// TIA Portal project "trietRot_Nhat" (V16)

(* hardware
DEVICE "S7-1200 station_1"  S7-1200 Station
   slot 0: "Rack_0"  S7-1200 Rack  Rack  V1.0
   slot 1: "PLC_1"  CPU 1214C AC/DC/Rly  6ES7 214-1BG40-0XB0  V4.4
*)

// ===== PLC "PLC_1"  CPU 1214C AC/DC/Rly =====

VAR_GLOBAL   // PLC tag table "Default tag table"
   "START" AT %M6.0 : Bool;
   "AUTO" AT %M6.1 : Bool;
   "TG1" AT %M1.1 : Bool;
   "TG2" AT %M1.2 : Bool;
   "STOP" AT %M6.2 : Bool;
   "Đèn" AT %Q0.0 : Bool;
   "Băng tải 2" AT %Q0.2 : Bool;
   "Tag_1" AT %M2.0 : Bool;
   "CB4" AT %M2.4 : Bool;
   "Băng tải 1" AT %Q0.1 : Bool;
   "CB3" AT %M2.3 : Bool;
   "Tag_2" AT %MD10 : DWord;
   "Tag_3" AT %M3.0 : Bool;
   "Sản phẩm hiện tại" AT %MW10 : Int;
   "Thiết lập số sản phẩm trong thùng" AT %MW20 : Int;
   "CB1" AT %M2.1 : Bool;
   "CB2" AT %M2.2 : Bool;
   "Bơm" AT %Q0.3 : Bool;
   "Van" AT %Q0.4 : Bool;
   "Clock_Byte" AT %MB0 : Byte;
   "Clock_2Hz" AT %M0.3 : Bool;
   "Clock_1.25Hz" AT %M0.4 : Bool;
   "Clock_1Hz" AT %M0.5 : Bool;
   "Clock_0.625Hz" AT %M0.6 : Bool;
   "Clock_0.5Hz" AT %M0.7 : Bool;
   "Tag_5" AT %M10.0 : Bool;
   "Giá trị lượng nước hiện tại" AT %MW40 : Int;
   "Thiết lập lượng nước cần rót" AT %MW30 : Int;
   "Xilanh1" AT %Q0.5 : Bool;
   "Xilanh2" AT %Q0.6 : Bool;
   "Thiết lập số thùng hàng" AT %MW50 : Int;
   "Số thùng hàng hiện tại" AT %MW60 : Int;
   "TG3" AT %M1.3 : Bool;
   "TG4" AT %M1.4 : Bool;
   "Tag_4" AT %M1.5 : Bool;
   "Tag_6" AT %MW100 : Int;
   "Tag_7" AT %M1.6 : Bool;
   "CB5" AT %M2.5 : Bool;
   "Tag_9" AT %M11.0 : Bool;
   "Tag_10" AT %M11.1 : Bool;
   "Tag_11" AT %M12.0 : Bool;
   "Tag_12" AT %M12.1 : Bool;
END_VAR

// folder: System blocks/Program resources

DATA_BLOCK "IEC_Counter_0_DB"   // DB1
{ S7_Optimized_Access := 'TRUE' }
AUTHOR : Simatic
FAMILY : IEC
NAME : CNTR
VERSION : 1.0
// stored: InstanceOfName IEC_COUNTER
"IEC_COUNTER"
BEGIN
END_DATA_BLOCK

DATA_BLOCK "T1"   // DB2
{ S7_Optimized_Access := 'TRUE' }
AUTHOR : Simatic
FAMILY : IEC
NAME : IEC_TMR
VERSION : 1.0
// stored: InstanceOfName IEC_TIMER
"IEC_TIMER"
BEGIN
END_DATA_BLOCK

DATA_BLOCK "CTU"   // DB3
{ S7_Optimized_Access := 'TRUE' }
AUTHOR : Simatic
FAMILY : IEC
NAME : CNTR
VERSION : 1.0
// stored: InstanceOfName IEC_COUNTER
"IEC_COUNTER"
BEGIN
END_DATA_BLOCK

DATA_BLOCK "t3"   // DB5
{ S7_Optimized_Access := 'TRUE' }
AUTHOR : Simatic
FAMILY : IEC
NAME : IEC_TMR
VERSION : 1.0
// stored: InstanceOfName IEC_TIMER
"IEC_TIMER"
BEGIN
END_DATA_BLOCK

// folder: (top level)

ORGANIZATION_BLOCK "Main"   // OB1, LAD, ProgramCycle
TITLE = "Main Program Sweep (Cycle)"
{ S7_Optimized_Access := 'TRUE' }
VERSION : 0.1
   VAR_INPUT
      Initial_Call : Bool;   // Initial call of this OB
      Remanence : Bool;   // =True, if remanent data are available
   END_VAR
   VAR_TEMP   // added for the SCL form of the ladder/FBD networks
      _w1 : Bool;
      _w2 : Bool;
      _w3 : Bool;
   END_VAR
BEGIN

REGION Network 1
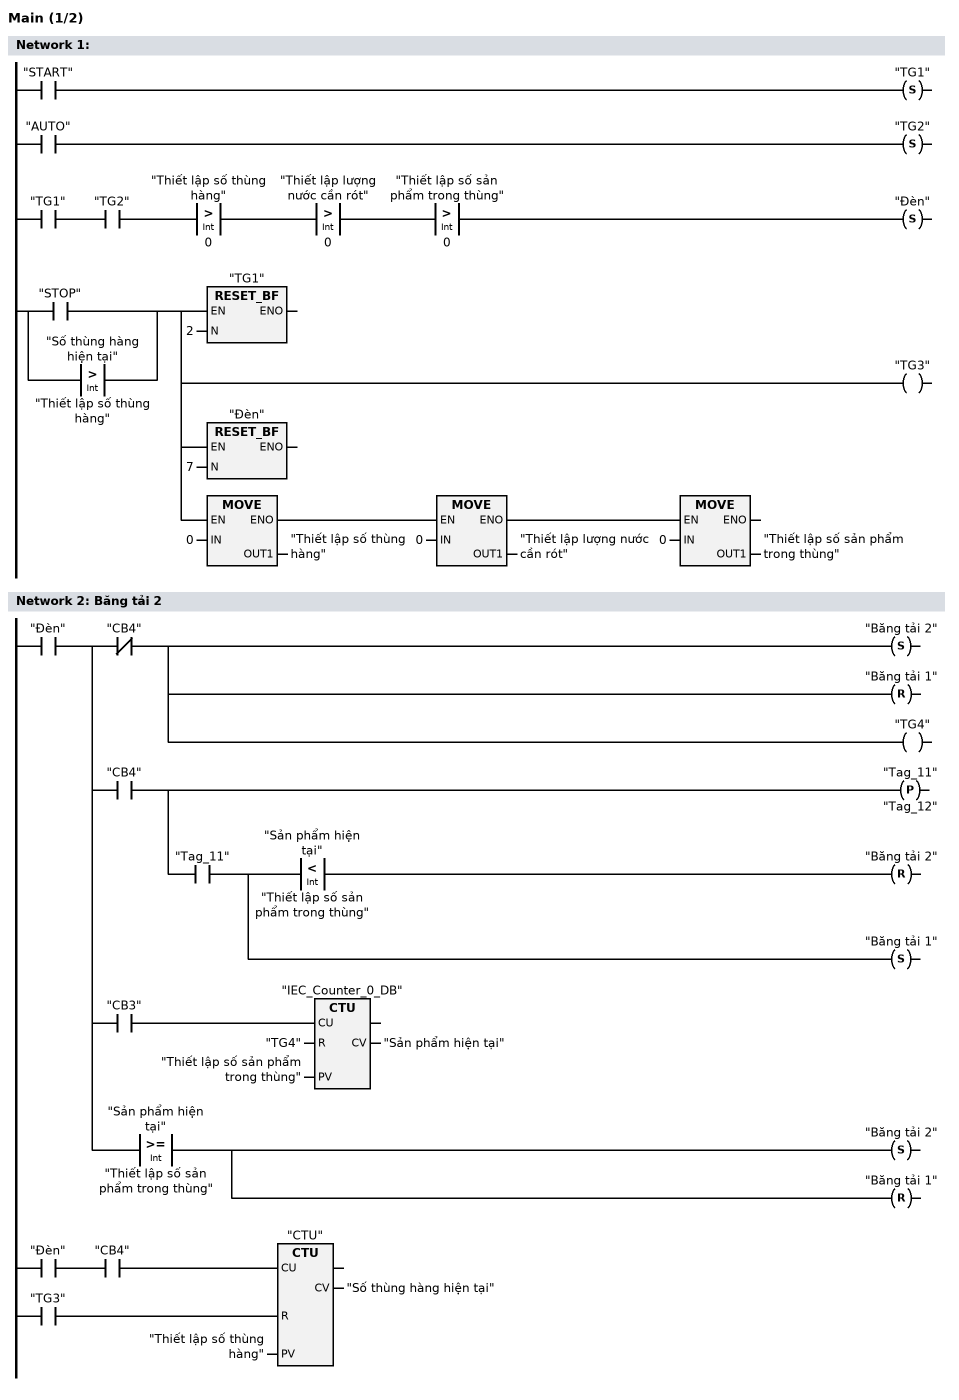
   // no SCL statement known for RBitfield: written as a call
   IF "START" THEN "TG1" := TRUE; END_IF;
   IF "AUTO" THEN "TG2" := TRUE; END_IF;
   IF "TG1" AND "TG2" AND ("Thiết lập số thùng hàng" > 0) AND ("Thiết lập lượng nước cần rót" > 0) AND ("Thiết lập số sản phẩm trong thùng" > 0) THEN
       "Đèn" := TRUE;
   END_IF;
   #_w1 := "STOP" OR ("Số thùng hàng hiện tại" > "Thiết lập số thùng hàng");
   IF #_w1 THEN RESET_BF(operand := "TG1", n := 2); END_IF;
   "TG3" := #_w1;
   IF #_w1 THEN
       RESET_BF(operand := "Đèn", n := 7);
       "Thiết lập số thùng hàng" := 0;
       "Thiết lập lượng nước cần rót" := 0;
       "Thiết lập số sản phẩm trong thùng" := 0;
   END_IF;
END_REGION

REGION Network 2: Băng tải 2
   #_w1 := "Đèn" AND NOT "CB4";
   IF #_w1 THEN
       "Băng tải 2" := TRUE;
       "Băng tải 1" := FALSE;
   END_IF;
   "TG4" := #_w1;
   #_w2 := "Đèn" AND "CB4";
   "Tag_11" := #_w2 AND NOT "Tag_12";   // rising edge
   "Tag_12" := #_w2;
   #_w3 := #_w2 AND "Tag_11";
   IF #_w3 AND ("Sản phẩm hiện tại" < "Thiết lập số sản phẩm trong thùng") THEN
       "Băng tải 2" := FALSE;
   END_IF;
   IF #_w3 THEN "Băng tải 1" := TRUE; END_IF;
   "IEC_Counter_0_DB".CTU(CU := "Đèn" AND "CB3",
                          R := "TG4",
                          PV := "Thiết lập số sản phẩm trong thùng",
                          CV => "Sản phẩm hiện tại");
   IF "Đèn" AND ("Sản phẩm hiện tại" >= "Thiết lập số sản phẩm trong thùng") THEN
       "Băng tải 2" := TRUE;
       "Băng tải 1" := FALSE;
   END_IF;
   "CTU".CTU(CU := "Đèn" AND "CB4", R := "TG3", PV := "Thiết lập số thùng hàng", CV => "Số thùng hàng hiện tại");
END_REGION

REGION Network 3: Băng tải 1
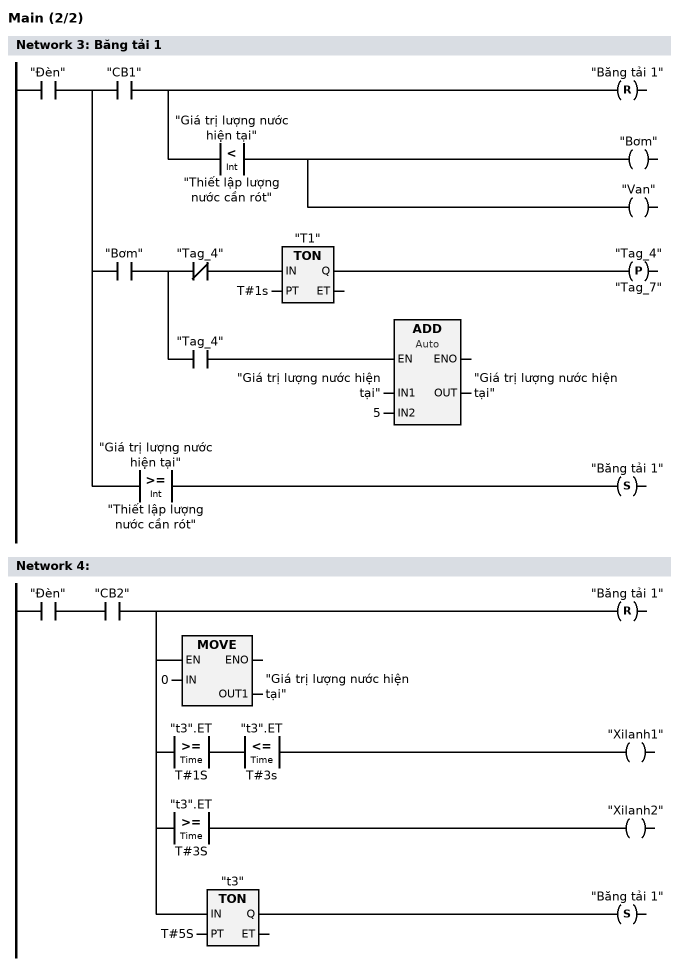
   #_w1 := "Đèn" AND "CB1";
   IF #_w1 THEN "Băng tải 1" := FALSE; END_IF;
   "Bơm" := #_w1 AND ("Giá trị lượng nước hiện tại" < "Thiết lập lượng nước cần rót");
   "Van" := "Bơm";
   #_w2 := "Đèn" AND "Bơm";
   "T1".TON(IN := #_w2 AND NOT "Tag_4", PT := T#1s);
   "Tag_4" := "T1".Q AND NOT "Tag_7";   // rising edge
   "Tag_7" := "T1".Q;
   IF #_w2 AND "Tag_4" THEN "Giá trị lượng nước hiện tại" := "Giá trị lượng nước hiện tại" + 5; END_IF;
   IF "Đèn" AND ("Giá trị lượng nước hiện tại" >= "Thiết lập lượng nước cần rót") THEN
       "Băng tải 1" := TRUE;
   END_IF;
END_REGION

REGION Network 4
   #_w1 := "Đèn" AND "CB2";
   IF #_w1 THEN
       "Băng tải 1" := FALSE;
       "Giá trị lượng nước hiện tại" := 0;
   END_IF;
   "Xilanh1" := #_w1 AND ("t3".ET >= T#1S) AND ("t3".ET <= T#3s);
   "Xilanh2" := #_w1 AND ("t3".ET >= T#3S);
   "t3".TON(IN := #_w1, PT := T#5S);
   IF "t3".Q THEN "Băng tải 1" := TRUE; END_IF;
END_REGION
END_ORGANIZATION_BLOCK